FUNCTION_BLOCK ERODE (* openCV erode filter *)
  (* Version 1.0, AN, SWDC RTSoft *)
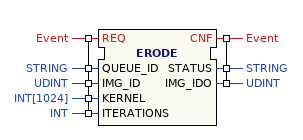
  EVENT_INPUT
    REQ WITH QUEUE_ID, IMG_ID, KERNEL, ITERATIONS;
  END_EVENT
  EVENT_OUTPUT
    CNF WITH STATUS, IMG_IDO;
  END_EVENT
  VAR_INPUT
    QUEUE_ID : STRING;
    IMG_ID : UDINT;
    KERNEL : ARRAY [0..1023] OF INT; (* Erosion kernel. Array of integers will be reshaped into a square matrix *)
    ITERATIONS : INT;
  END_VAR
  VAR_OUTPUT
    STATUS : STRING;
    IMG_IDO : UDINT;
  END_VAR
  ALGORITHM REQ IN ST:

  END_ALGORITHM
END_FUNCTION_BLOCK
